(* Logix 5000 project; controller SX_V040001_C001 vendor 1 type 14 code 77 rev 16.22; software revision 16.04; part 34 of 35 *)
(* tags used below, declared in another part *)
   ALL_KINDS : INT[90];
   Basic : INT;
   C_MINUTES : COUNTER;
   C_SECONDS : COUNTER;
   choco_control : PID;
   G_AInput : DINT[8];
   G_AOutput : DINT[8];
   G_DInput : DINT[3];
   G_DOutput : DINT[3];
   M_VKE_1 : BOOL;
   mw_temp : DINT;
   PARAMETER : INT[501];
   REMOTE_DATA_IN : INT[510];
   REMOTE_DATA_OUT : INT[510];
   REMOTE_SYSTEM : INT[38];
   T_COOLING_VALVE : TIMER;
   T_HEATING_VALVE : TIMER;
   TEMP : INT[14];
   TEMP_REAL : REAL[22];
   TIMER_CHOCO_CONTR : TIMER;
   TIMER_WATER_CONTR : TIMER;
   water_control : PID;
(* MainProgram, continued *)

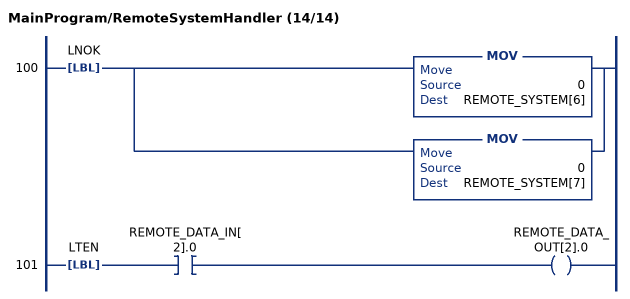
   [picture p744: MainProgram/RemoteSystemHandler rungs 100-101]
   100: LBL(LNOK)[MOV(0,REMOTE_SYSTEM[6]) ,MOV(0,REMOTE_SYSTEM[7]) ];
   101: LBL(LTEN)XIC(REMOTE_DATA_IN[2].0)OTE(REMOTE_DATA_OUT[2].0);
END_ROUTINE

ROUTINE Simulator   (* ladder *)
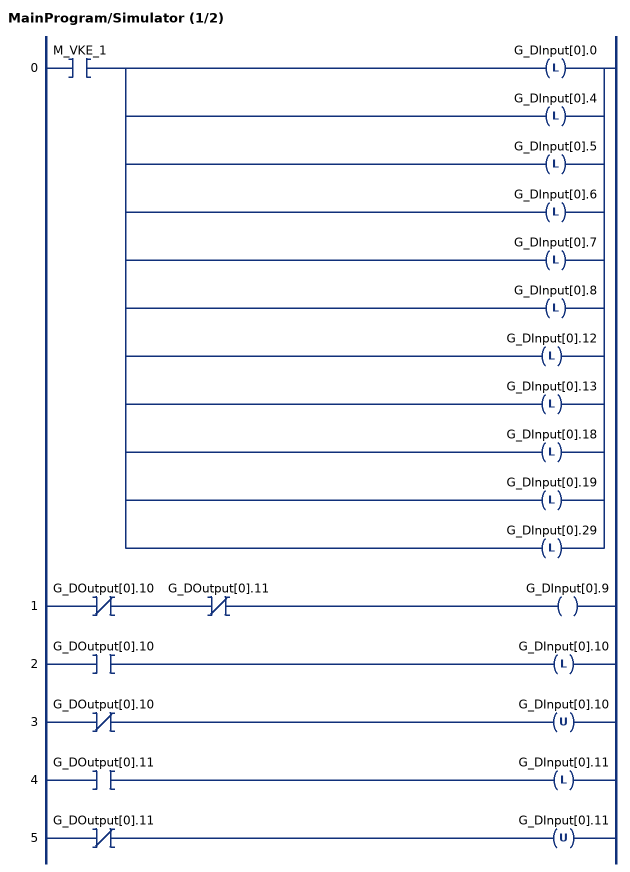
   0: XIC(M_VKE_1)[OTL(G_DInput[0].0) ,OTL(G_DInput[0].4) ,OTL(G_DInput[0].5) ,OTL(G_DInput[0].6) ,OTL(G_DInput[0].7) ,OTL(G_DInput[0].8) ,OTL(G_DInput[0].12) ,OTL(G_DInput[0].13) ,OTL(G_DInput[0].18) ,OTL(G_DInput[0].19) ,OTL(G_DInput[0].29) ];
   1: XIO(G_DOutput[0].10)XIO(G_DOutput[0].11)OTE(G_DInput[0].9);
   2: XIC(G_DOutput[0].10)OTL(G_DInput[0].10);
   3: XIO(G_DOutput[0].10)OTU(G_DInput[0].10);
   4: XIC(G_DOutput[0].11)OTL(G_DInput[0].11);
   5: XIO(G_DOutput[0].11)OTU(G_DInput[0].11);
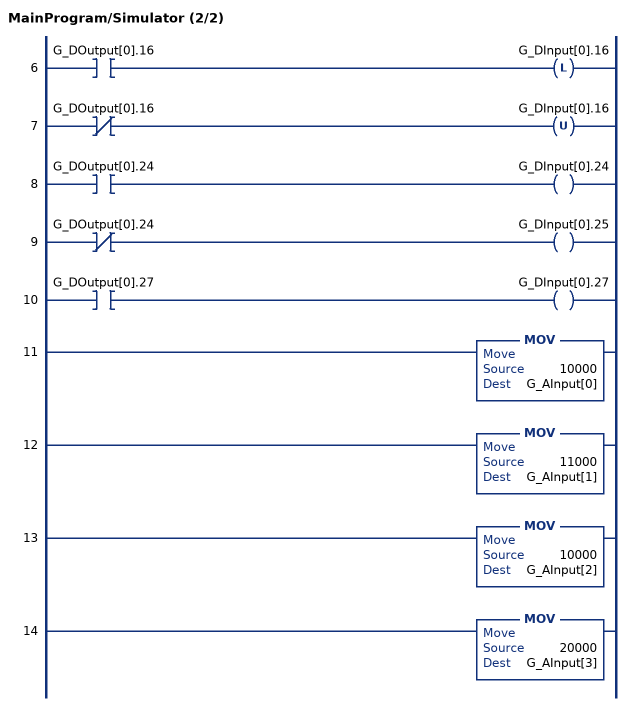
   6: XIC(G_DOutput[0].16)OTL(G_DInput[0].16);
   7: XIO(G_DOutput[0].16)OTU(G_DInput[0].16);
   8: XIC(G_DOutput[0].24)OTE(G_DInput[0].24);
   9: XIO(G_DOutput[0].24)OTE(G_DInput[0].25);
   10: XIC(G_DOutput[0].27)OTE(G_DInput[0].27);
   11: MOV(10000,G_AInput[0]);
   12: MOV(11000,G_AInput[1]);
   13: MOV(10000,G_AInput[2]);
   14: MOV(20000,G_AInput[3]);
END_ROUTINE

ROUTINE SSW_Signals   (* ladder *)
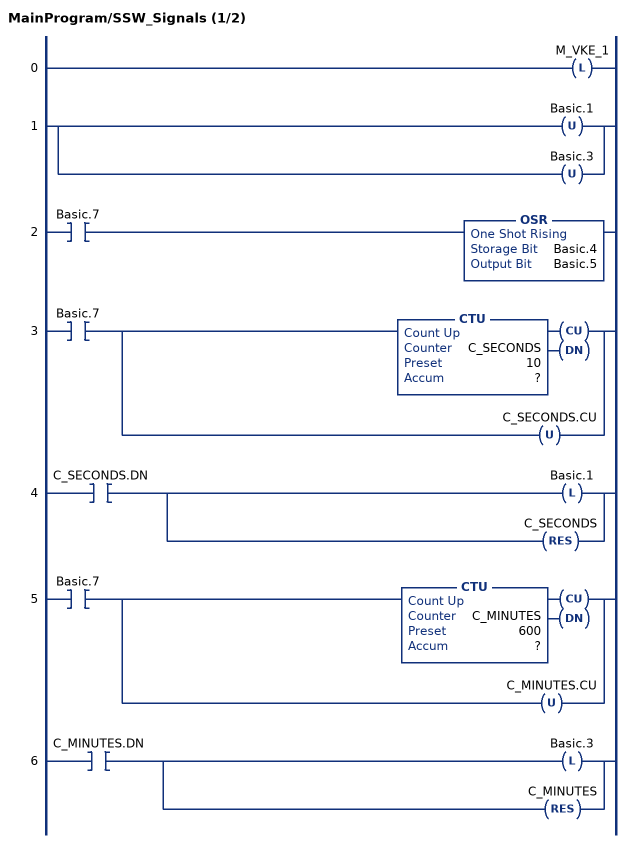
   0: OTL(M_VKE_1);
   1: [OTU(Basic.1) ,OTU(Basic.3) ];
   2: XIC(Basic.7)OSR(Basic.4,Basic.5);
   3: XIC(Basic.7)[CTU(C_SECONDS,?,?) ,OTU(C_SECONDS.CU) ];
   4: XIC(C_SECONDS.DN)[OTL(Basic.1) ,RES(C_SECONDS) ];
   5: XIC(Basic.7)[CTU(C_MINUTES,?,?) ,OTU(C_MINUTES.CU) ];
   6: XIC(C_MINUTES.DN)[OTL(Basic.3) ,RES(C_MINUTES) ];
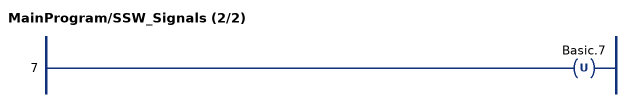
   7: OTU(Basic.7);
END_ROUTINE

ROUTINE TempControl   (* ladder *)
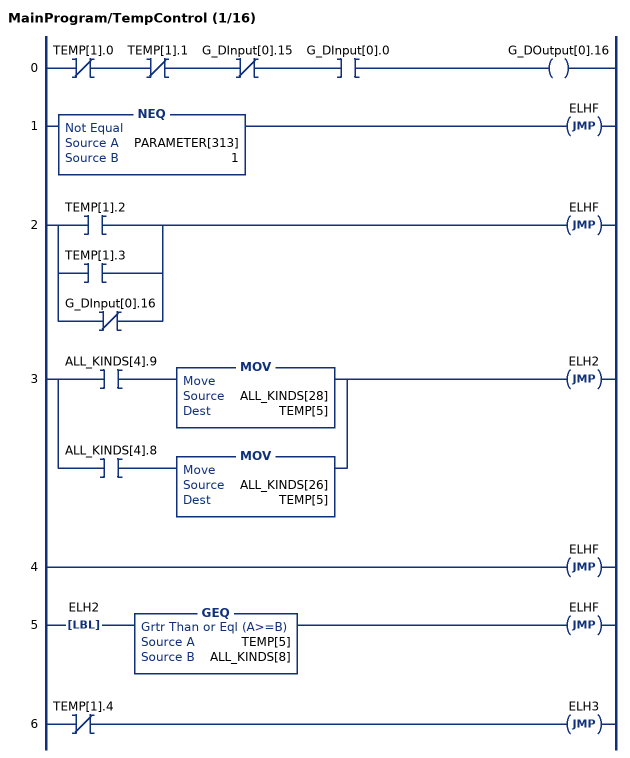
   0: XIO(TEMP[1].0)XIO(TEMP[1].1)XIO(G_DInput[0].15)XIC(G_DInput[0].0)OTE(G_DOutput[0].16);
   1: NEQ(PARAMETER[313],1)JMP(ELHF);
   2: [XIC(TEMP[1].2) ,XIC(TEMP[1].3) ,XIO(G_DInput[0].16) ]JMP(ELHF);
   3: [XIC(ALL_KINDS[4].9) MOV(ALL_KINDS[28],TEMP[5]) ,XIC(ALL_KINDS[4].8) MOV(ALL_KINDS[26],TEMP[5]) ]JMP(ELH2);
   4: JMP(ELHF);
   5: LBL(ELH2)GEQ(TEMP[5],ALL_KINDS[8])JMP(ELHF);
   6: XIO(TEMP[1].4)JMP(ELH3);
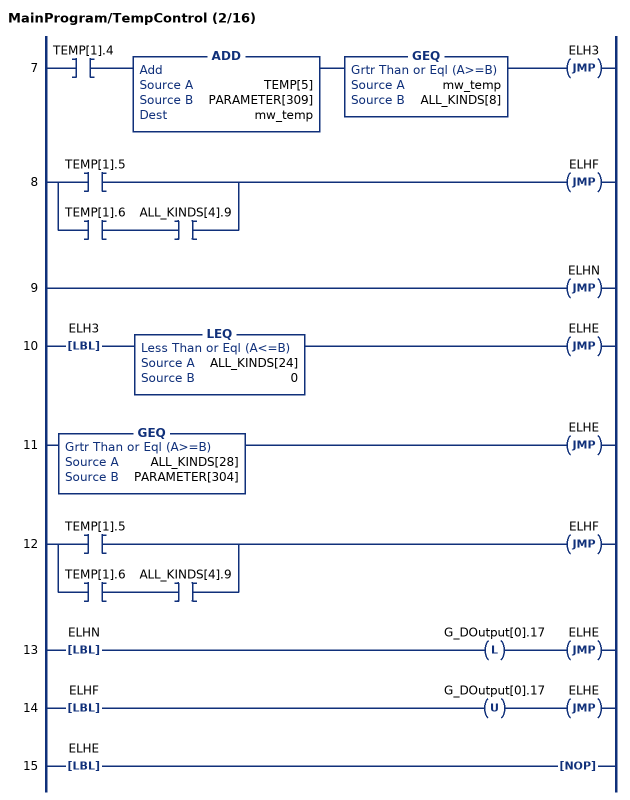
   7: XIC(TEMP[1].4)ADD(TEMP[5],PARAMETER[309],mw_temp)GEQ(mw_temp,ALL_KINDS[8])JMP(ELH3);
   8: [XIC(TEMP[1].5) ,XIC(TEMP[1].6) XIC(ALL_KINDS[4].9) ]JMP(ELHF);
   9: JMP(ELHN);
   10: LBL(ELH3)LEQ(ALL_KINDS[24],0)JMP(ELHE);
   11: GEQ(ALL_KINDS[28],PARAMETER[304])JMP(ELHE);
   12: [XIC(TEMP[1].5) ,XIC(TEMP[1].6) XIC(ALL_KINDS[4].9) ]JMP(ELHF);
   13: LBL(ELHN)OTL(G_DOutput[0].17)JMP(ELHE);
   14: LBL(ELHF)OTU(G_DOutput[0].17)JMP(ELHE);
   15: LBL(ELHE)NOP();
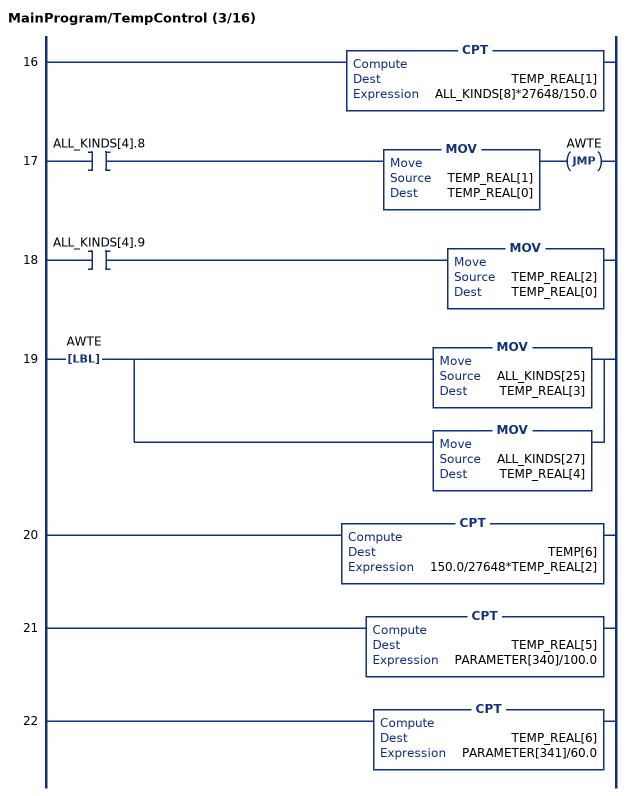
   16: CPT(TEMP_REAL[1],ALL_KINDS[8]*27648/150.0);
   17: XIC(ALL_KINDS[4].8)MOV(TEMP_REAL[1],TEMP_REAL[0])JMP(AWTE);
   18: XIC(ALL_KINDS[4].9)MOV(TEMP_REAL[2],TEMP_REAL[0]);
   19: LBL(AWTE)[MOV(ALL_KINDS[25],TEMP_REAL[3]) ,MOV(ALL_KINDS[27],TEMP_REAL[4]) ];
   20: CPT(TEMP[6],150.0/27648*TEMP_REAL[2]);
   21: CPT(TEMP_REAL[5],PARAMETER[340]/100.0);
   22: CPT(TEMP_REAL[6],PARAMETER[341]/60.0);
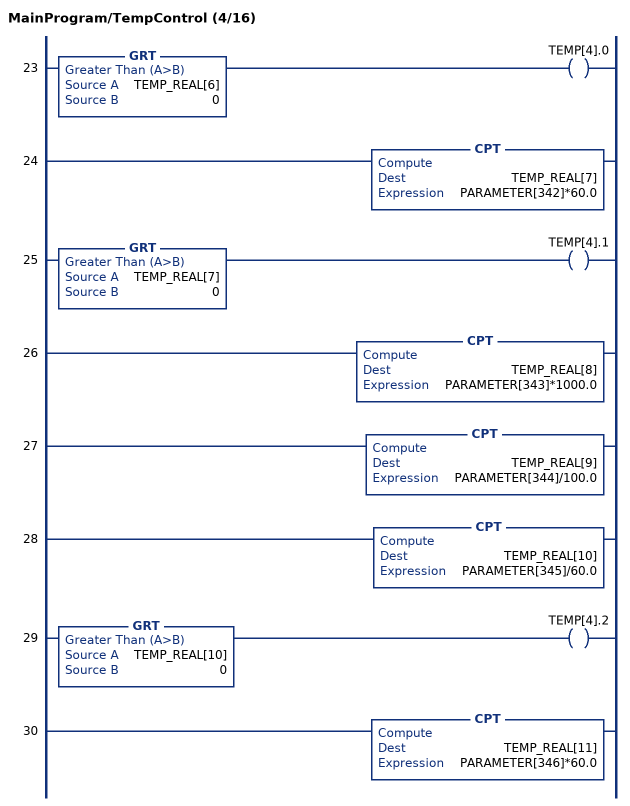
   23: GRT(TEMP_REAL[6],0)OTE(TEMP[4].0);
   24: CPT(TEMP_REAL[7],PARAMETER[342]*60.0);
   25: GRT(TEMP_REAL[7],0)OTE(TEMP[4].1);
   26: CPT(TEMP_REAL[8],PARAMETER[343]*1000.0);
   27: CPT(TEMP_REAL[9],PARAMETER[344]/100.0);
   28: CPT(TEMP_REAL[10],PARAMETER[345]/60.0);
   29: GRT(TEMP_REAL[10],0)OTE(TEMP[4].2);
   30: CPT(TEMP_REAL[11],PARAMETER[346]*60.0);
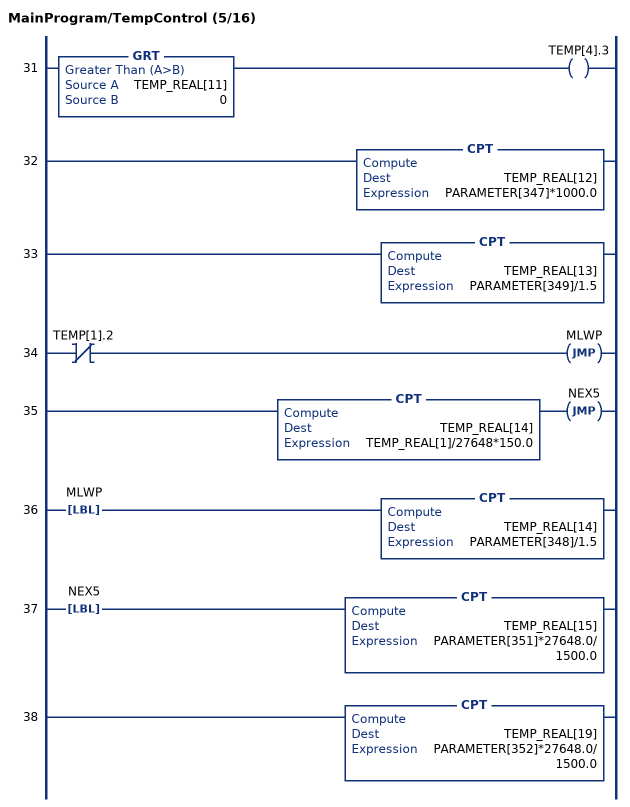
   31: GRT(TEMP_REAL[11],0)OTE(TEMP[4].3);
   32: CPT(TEMP_REAL[12],PARAMETER[347]*1000.0);
   33: CPT(TEMP_REAL[13],PARAMETER[349]/1.5);
   34: XIO(TEMP[1].2)JMP(MLWP);
   35: CPT(TEMP_REAL[14],TEMP_REAL[1]/27648*150.0)JMP(NEX5);
   36: LBL(MLWP)CPT(TEMP_REAL[14],PARAMETER[348]/1.5);
   37: LBL(NEX5)CPT(TEMP_REAL[15],PARAMETER[351]*27648.0/1500.0);
   38: CPT(TEMP_REAL[19],PARAMETER[352]*27648.0/1500.0);
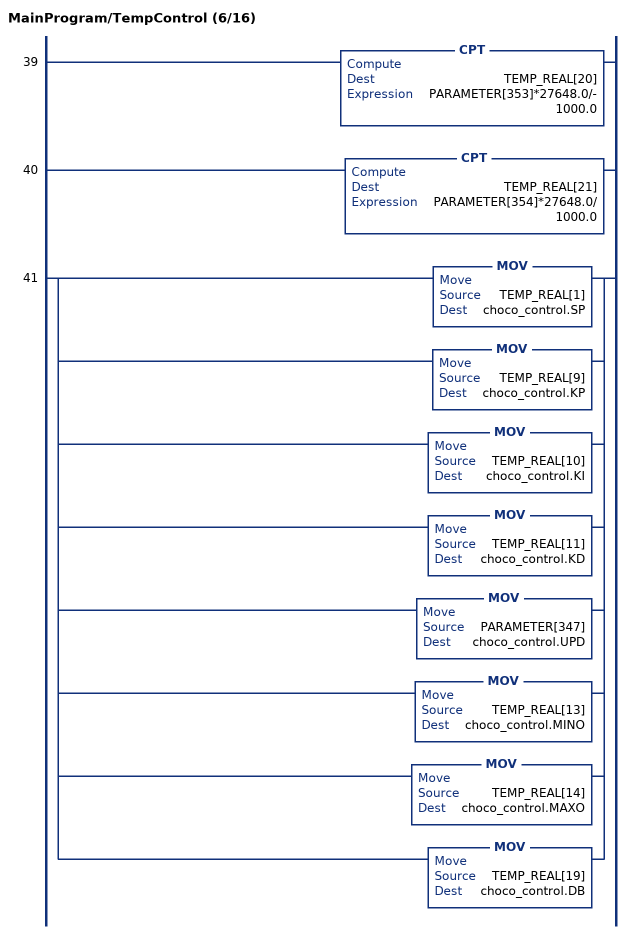
   39: CPT(TEMP_REAL[20],PARAMETER[353]*27648.0/-1000.0);
   40: CPT(TEMP_REAL[21],PARAMETER[354]*27648.0/1000.0);
   41: [MOV(TEMP_REAL[1],choco_control.SP) ,MOV(TEMP_REAL[9],choco_control.KP) ,MOV(TEMP_REAL[10],choco_control.KI) ,MOV(TEMP_REAL[11],choco_control.KD) ,MOV(PARAMETER[347],choco_control.UPD) ,MOV(TEMP_REAL[13],choco_control.MINO) ,MOV(TEMP_REAL[14],choco_control.MAXO) ,MOV(TEMP_REAL[19],choco_control.DB) ];
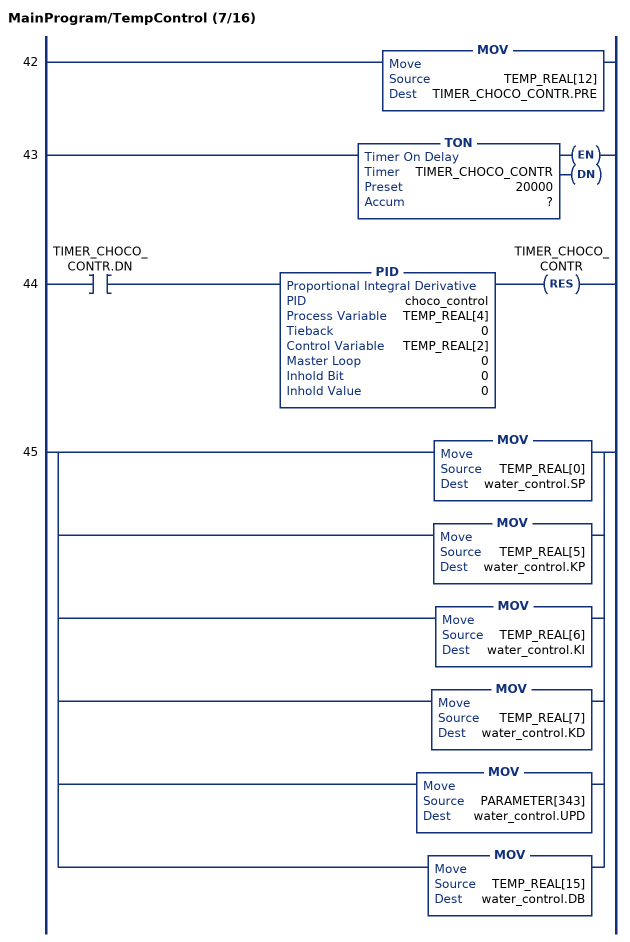
   42: MOV(TEMP_REAL[12],TIMER_CHOCO_CONTR.PRE);
   43: TON(TIMER_CHOCO_CONTR,?,?);
   44: XIC(TIMER_CHOCO_CONTR.DN)PID(choco_control,TEMP_REAL[4],0,TEMP_REAL[2],0,0,0)RES(TIMER_CHOCO_CONTR);
   45: [MOV(TEMP_REAL[0],water_control.SP) ,MOV(TEMP_REAL[5],water_control.KP) ,MOV(TEMP_REAL[6],water_control.KI) ,MOV(TEMP_REAL[7],water_control.KD) ,MOV(PARAMETER[343],water_control.UPD) ,MOV(TEMP_REAL[15],water_control.DB) ];
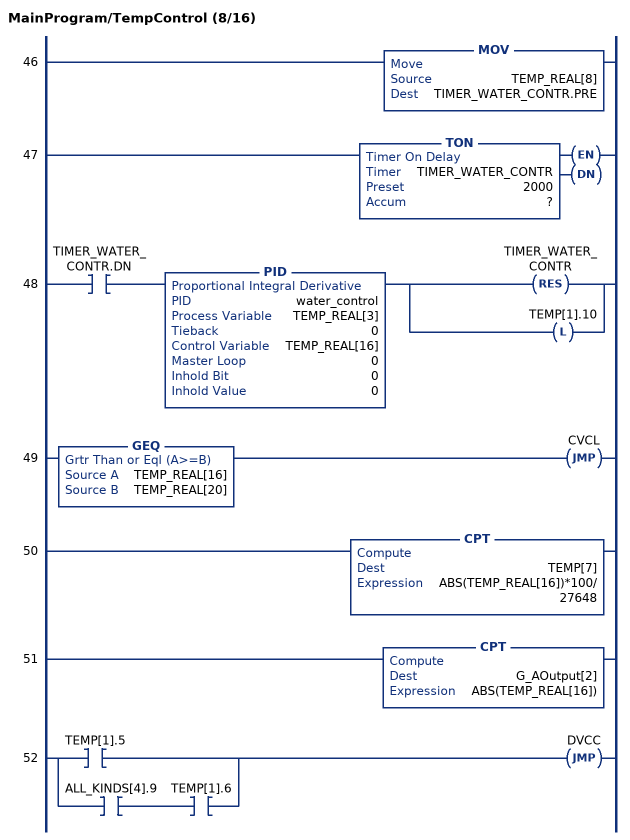
   46: MOV(TEMP_REAL[8],TIMER_WATER_CONTR.PRE);
   47: TON(TIMER_WATER_CONTR,?,?);
   48: XIC(TIMER_WATER_CONTR.DN)PID(water_control,TEMP_REAL[3],0,TEMP_REAL[16],0,0,0)[RES(TIMER_WATER_CONTR) ,OTL(TEMP[1].10) ];
   49: GEQ(TEMP_REAL[16],TEMP_REAL[20])JMP(CVCL);
   50: CPT(TEMP[7],ABS(TEMP_REAL[16])*100/27648);
   51: CPT(G_AOutput[2],ABS(TEMP_REAL[16]));
   52: [XIC(TEMP[1].5) ,XIC(ALL_KINDS[4].9) XIC(TEMP[1].6) ]JMP(DVCC);
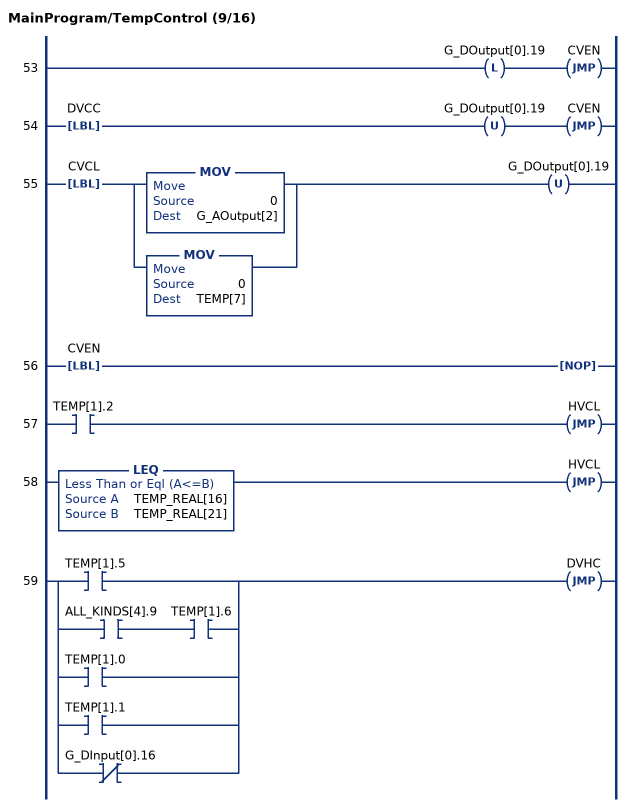
   53: OTL(G_DOutput[0].19)JMP(CVEN);
   54: LBL(DVCC)OTU(G_DOutput[0].19)JMP(CVEN);
   55: LBL(CVCL)[MOV(0,G_AOutput[2]) ,MOV(0,TEMP[7]) ]OTU(G_DOutput[0].19);
   56: LBL(CVEN)NOP();
   57: XIC(TEMP[1].2)JMP(HVCL);
   58: LEQ(TEMP_REAL[16],TEMP_REAL[21])JMP(HVCL);
   59: [XIC(TEMP[1].5) ,XIC(ALL_KINDS[4].9) XIC(TEMP[1].6) ,XIC(TEMP[1].0) ,XIC(TEMP[1].1) ,XIO(G_DInput[0].16) ]JMP(DVHC);
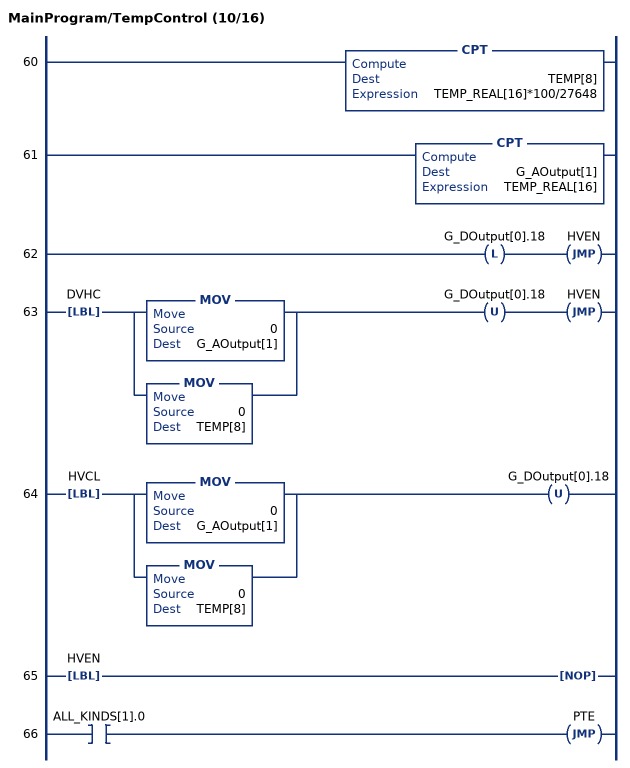
   60: CPT(TEMP[8],TEMP_REAL[16]*100/27648);
   61: CPT(G_AOutput[1],TEMP_REAL[16]);
   62: OTL(G_DOutput[0].18)JMP(HVEN);
   63: LBL(DVHC)[MOV(0,G_AOutput[1]) ,MOV(0,TEMP[8]) ]OTU(G_DOutput[0].18)JMP(HVEN);
   64: LBL(HVCL)[MOV(0,G_AOutput[1]) ,MOV(0,TEMP[8]) ]OTU(G_DOutput[0].18);
   65: LBL(HVEN)NOP();
   66: XIC(ALL_KINDS[1].0)JMP(PTE);
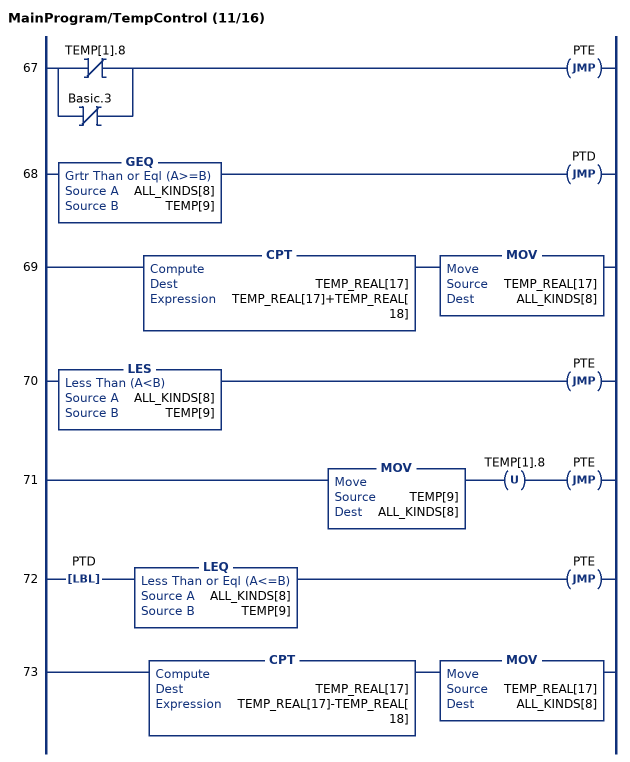
   67: [XIO(TEMP[1].8) ,XIO(Basic.3) ]JMP(PTE);
   68: GEQ(ALL_KINDS[8],TEMP[9])JMP(PTD);
   69: CPT(TEMP_REAL[17],TEMP_REAL[17]+TEMP_REAL[18])MOV(TEMP_REAL[17],ALL_KINDS[8]);
   70: LES(ALL_KINDS[8],TEMP[9])JMP(PTE);
   71: MOV(TEMP[9],ALL_KINDS[8])OTU(TEMP[1].8)JMP(PTE);
   72: LBL(PTD)LEQ(ALL_KINDS[8],TEMP[9])JMP(PTE);
   73: CPT(TEMP_REAL[17],TEMP_REAL[17]-TEMP_REAL[18])MOV(TEMP_REAL[17],ALL_KINDS[8]);
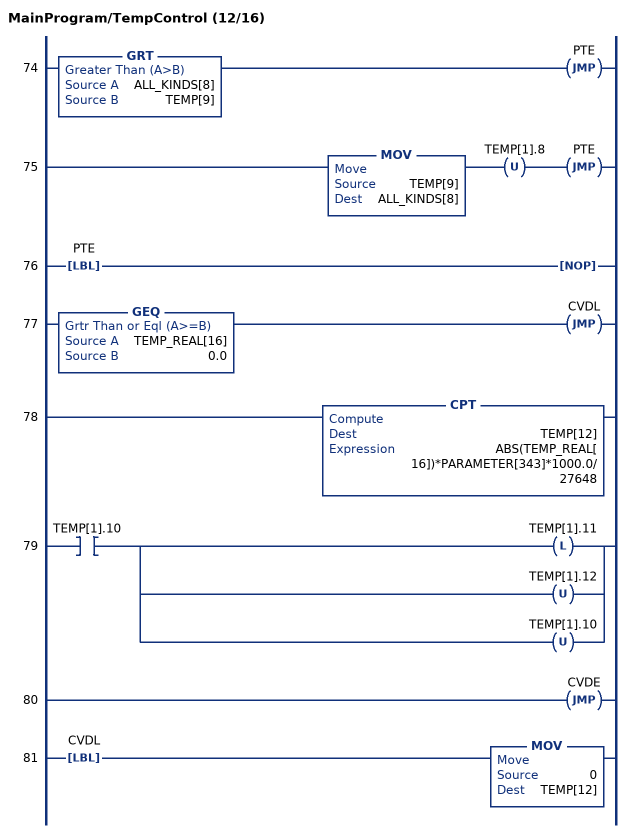
   74: GRT(ALL_KINDS[8],TEMP[9])JMP(PTE);
   75: MOV(TEMP[9],ALL_KINDS[8])OTU(TEMP[1].8)JMP(PTE);
   76: LBL(PTE)NOP();
   77: GEQ(TEMP_REAL[16],0.0)JMP(CVDL);
   78: CPT(TEMP[12],ABS(TEMP_REAL[16])*PARAMETER[343]*1000.0/27648);
   79: XIC(TEMP[1].10)[OTL(TEMP[1].11) ,OTU(TEMP[1].12) ,OTU(TEMP[1].10) ];
   80: JMP(CVDE);
   81: LBL(CVDL)MOV(0,TEMP[12]);
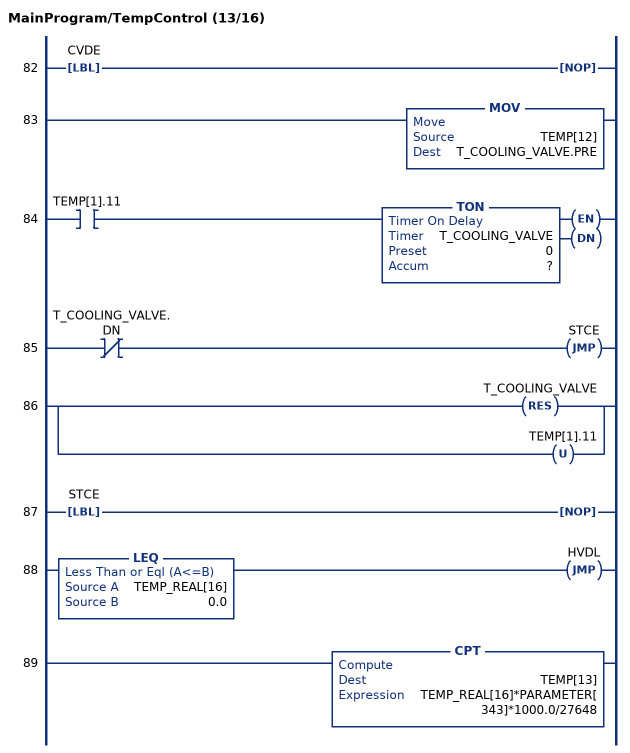
   82: LBL(CVDE)NOP();
   83: MOV(TEMP[12],T_COOLING_VALVE.PRE);
   84: XIC(TEMP[1].11)TON(T_COOLING_VALVE,?,?);
   85: XIO(T_COOLING_VALVE.DN)JMP(STCE);
   86: [RES(T_COOLING_VALVE) ,OTU(TEMP[1].11) ];
   87: LBL(STCE)NOP();
   88: LEQ(TEMP_REAL[16],0.0)JMP(HVDL);
   89: CPT(TEMP[13],TEMP_REAL[16]*PARAMETER[343]*1000.0/27648);
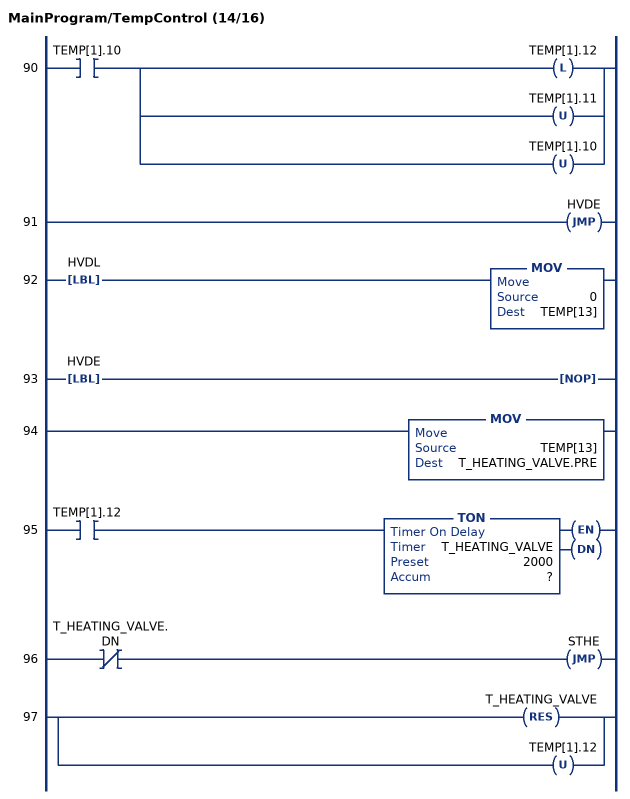
   90: XIC(TEMP[1].10)[OTL(TEMP[1].12) ,OTU(TEMP[1].11) ,OTU(TEMP[1].10) ];
   91: JMP(HVDE);
   92: LBL(HVDL)MOV(0,TEMP[13]);
   93: LBL(HVDE)NOP();
   94: MOV(TEMP[13],T_HEATING_VALVE.PRE);
   95: XIC(TEMP[1].12)TON(T_HEATING_VALVE,?,?);
   96: XIO(T_HEATING_VALVE.DN)JMP(STHE);
   97: [RES(T_HEATING_VALVE) ,OTU(TEMP[1].12) ];
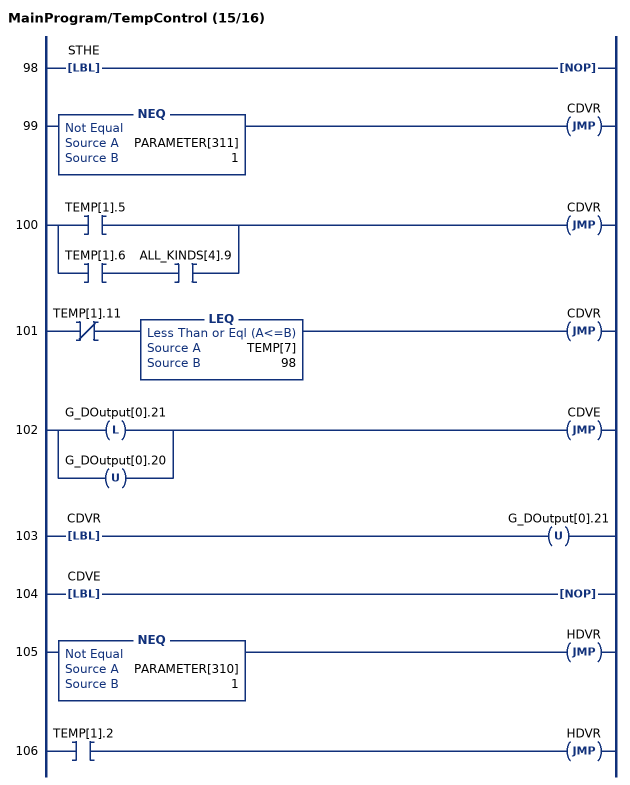
   98: LBL(STHE)NOP();
   99: NEQ(PARAMETER[311],1)JMP(CDVR);
   100: [XIC(TEMP[1].5) ,XIC(TEMP[1].6) XIC(ALL_KINDS[4].9) ]JMP(CDVR);
   101: XIO(TEMP[1].11)LEQ(TEMP[7],98)JMP(CDVR);
   102: [OTL(G_DOutput[0].21) ,OTU(G_DOutput[0].20) ]JMP(CDVE);
   103: LBL(CDVR)OTU(G_DOutput[0].21);
   104: LBL(CDVE)NOP();
   105: NEQ(PARAMETER[310],1)JMP(HDVR);
   106: XIC(TEMP[1].2)JMP(HDVR);
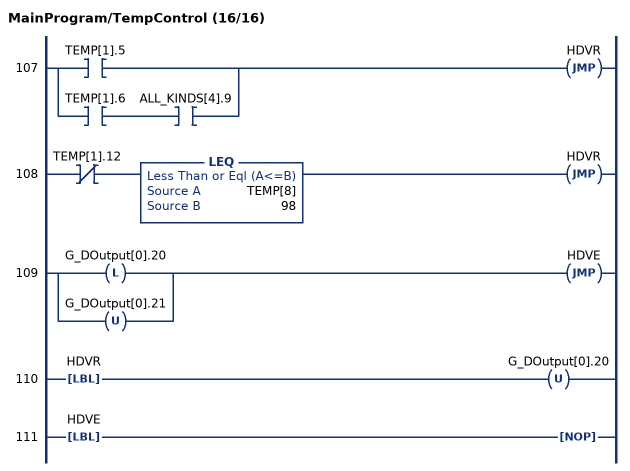
   107: [XIC(TEMP[1].5) ,XIC(TEMP[1].6) XIC(ALL_KINDS[4].9) ]JMP(HDVR);
   108: XIO(TEMP[1].12)LEQ(TEMP[8],98)JMP(HDVR);
   109: [OTL(G_DOutput[0].20) ,OTU(G_DOutput[0].21) ]JMP(HDVE);
   110: LBL(HDVR)OTU(G_DOutput[0].20);
   111: LBL(HDVE)NOP();
END_ROUTINE
